TYPE VECTOR_3 :
STRUCT
	X : REAL;
	Y : REAL;
	Z : REAL;
END_STRUCT
END_TYPE

(* stored: Version 1.1.0.1
   DUT VECTOR_3: Id {100d241d-2dd5-4bcc-bff0-3adf5a253b28} *)
